// TIA Portal V20 export
FUNCTION_BLOCK "FB_AxisPosition"   // FB411, SCL
{ S7_Optimized_Access := 'TRUE' }
// stored: AutoNumber false, MemoryReserve 100, SetENOAutomatically false
   VAR
      sError { ExternalAccessible := 'False'; ExternalVisible := 'False'; ExternalWritable := 'False'} : Bool;
      sNDR { ExternalAccessible := 'False'; ExternalVisible := 'False'; ExternalWritable := 'False'} : Bool;
      sState { ExternalAccessible := 'False'; ExternalVisible := 'False'; ExternalWritable := 'False'} : Word;
      sAxis01_X : Struct
         "$AA_IM" : LReal;
         "$MA_POS_LIMIT_MINUS" : LReal;
         "$MA_POS_LIMIT_MINUS2" : LReal;
         "$MA_POS_LIMIT_PLUS" : LReal;
         "$MA_POS_LIMIT_PLUS2" : LReal;
         "$MA_JOG_VELO" : LReal;
         "$MA_JOG_VELO_RAPID" : LReal;
         "$MA_MAX_AX_VELO" : LReal;
         "$A1_M_FP_POS4_30600" : LReal;
      END_STRUCT;
      sAxis02_Y : Struct
         "$AA_IM" : LReal;
         "$MA_POS_LIMIT_MINUS" : LReal;
         "$MA_POS_LIMIT_MINUS2" : LReal;
         "$MA_POS_LIMIT_PLUS" : LReal;
         "$MA_POS_LIMIT_PLUS2" : LReal;
         "$MA_JOG_VELO" : LReal;
         "$MA_JOG_VELO_RAPID" : LReal;
         "$MA_MAX_AX_VELO" : LReal;
      END_STRUCT;
      sAxis03_ZM : Struct
         "$AA_IM" : LReal;
         "$MA_POS_LIMIT_MINUS" : LReal;
         "$MA_POS_LIMIT_MINUS2" : LReal;
         "$MA_POS_LIMIT_PLUS" : LReal;
         "$MA_POS_LIMIT_PLUS2" : LReal;
         "$MA_JOG_VELO" : LReal;
         "$MA_JOG_VELO_RAPID" : LReal;
         "$MA_MAX_AX_VELO" : LReal;
      END_STRUCT;
      sAxis04_B : Struct
         "$AA_IM" : LReal;
         "$MA_POS_LIMIT_MINUS" : LReal;
         "$MA_POS_LIMIT_MINUS2" : LReal;
         "$MA_POS_LIMIT_PLUS" : LReal;
         "$MA_POS_LIMIT_PLUS2" : LReal;
         "$MA_JOG_VELO" : LReal;
         "$MA_JOG_VELO_RAPID" : LReal;
         "$MA_MAX_AX_VELO" : LReal;
      END_STRUCT;
      sAxis05_U1 : Struct
         "$AA_IM" : LReal;
         "$MA_POS_LIMIT_MINUS" : LReal;
         "$MA_POS_LIMIT_MINUS2" : LReal;
         "$MA_POS_LIMIT_PLUS" : LReal;
         "$MA_POS_LIMIT_PLUS2" : LReal;
         "$MA_JOG_VELO" : LReal;
         "$MA_JOG_VELO_RAPID" : LReal;
         "$MA_MAX_AX_VELO" : LReal;
      END_STRUCT;
      sAxis06_U2 : Struct
         "$AA_IM" : LReal;
         "$MA_POS_LIMIT_MINUS" : LReal;
         "$MA_POS_LIMIT_MINUS2" : LReal;
         "$MA_POS_LIMIT_PLUS" : LReal;
         "$MA_POS_LIMIT_PLUS2" : LReal;
         "$MA_JOG_VELO" : LReal;
         "$MA_JOG_VELO_RAPID" : LReal;
         "$MA_MAX_AX_VELO" : LReal;
         "$A1_M_FP_POS2_30600" : LReal;
      END_STRUCT;
      sAxis07_V : Struct
         "$AA_IM" : LReal;
         "$MA_POS_LIMIT_MINUS" : LReal;
         "$MA_POS_LIMIT_MINUS2" : LReal;
         "$MA_POS_LIMIT_PLUS" : LReal;
         "$MA_POS_LIMIT_PLUS2" : LReal;
         "$MA_JOG_VELO" : LReal;
         "$MA_JOG_VELO_RAPID" : LReal;
         "$MA_MAX_AX_VELO" : LReal;
      END_STRUCT;
      sAxis08_W : Struct
         "$AA_IM" : LReal;
         "$MA_POS_LIMIT_MINUS" : LReal;
         "$MA_POS_LIMIT_MINUS2" : LReal;
         "$MA_POS_LIMIT_PLUS" : LReal;
         "$MA_POS_LIMIT_PLUS2" : LReal;
         "$MA_JOG_VELO" : LReal;
         "$MA_JOG_VELO_RAPID" : LReal;
         "$MA_MAX_AX_VELO" : LReal;
      END_STRUCT;
      sAxis09_ZL : Struct
         "$AA_IM" : LReal;
         "$MA_POS_LIMIT_MINUS" : LReal;
         "$MA_POS_LIMIT_MINUS2" : LReal;
         "$MA_POS_LIMIT_PLUS" : LReal;
         "$MA_POS_LIMIT_PLUS2" : LReal;
         "$MA_JOG_VELO" : LReal;
         "$MA_JOG_VELO_RAPID" : LReal;
         "$MA_MAX_AX_VELO" : LReal;
      END_STRUCT;
   END_VAR
BEGIN
   REGION Description header 
       //==================================================================================
       // POSALUX Swiss SA / (C) Copyright 2025
       //----------------------------------------------------------------------------------
       // Title: FB_AxisPosition
       // Comment/Function: These function blocks allow reading NC data related to 
       //                   axis positions, references, and speeds from the NC.
       // Author: Fabien WALDT
       // Engineering: TIA Portal v17
       //----------------------------------------------------------------------------------
       // Change log table:
       // Version  | Date     | Expert in charge | Changes applied
       // ---------|----------|------------------|------------------------------------
       // 00.00.01 | 20250423 | WFA              | First released version
       // ==================================================================================
   END_REGION

   REGION Axis 01 X
       "LBP_ReadVar_DB_Axis01_X"(Req := "Clock_10Hz",
                                 NumVar := 8,
                                 Addr1 := "DB_NcVarSelect_AA_IM"."$AA_IM_Axis01_X".token,
                                 Addr2 := "DB_NcVarSelect_MA_POS_LIMIT_MINUS"."$MA_POS_LIMIT_MINUS_Axis01_X".token,
                                 Addr3 := "DB_NcVarSelect_MA_POS_LIMIT_MINUS2"."$MA_POS_LIMIT_MINUS2_Axis01_X".token,
                                 Addr4 := "DB_NcVarSelect_MA_POS_LIMIT_PLUS"."$MA_POS_LIMIT_PLUS_Axis01_X".token,
                                 Addr5 := "DB_NcVarSelect_MA_POS_LIMIT_PLUS2"."$MA_POS_LIMIT_PLUS2_Axis01_X".token,
                                 Addr6 := "DB_NcVarSelect_MA_JOG_VELO"."$MA_JOG_VELO_Axis01_X".token,
                                 Addr7 := "DB_NcVarSelect_MA_JOG_VELO_RAPID"."$MA_JOG_VELO_RAPID_Axis01_X".token,
                                 Addr8 := "DB_NcVarSelect_M_MAX_AX_VELO"."$MA_JOG_VELO_Axis01_X".token,
                                 Error => #sError,
                                 NDR => #sNDR,
                                 State => #sState,
                                 RD1 := #sAxis01_X."$AA_IM",
                                 RD2 := #sAxis01_X."$MA_POS_LIMIT_MINUS",
                                 RD3 := #sAxis01_X."$MA_POS_LIMIT_MINUS2",
                                 RD4 := #sAxis01_X."$MA_POS_LIMIT_PLUS",
                                 RD5 := #sAxis01_X."$MA_POS_LIMIT_PLUS2",
                                 RD6 := #sAxis01_X."$MA_JOG_VELO",
                                 RD7 := #sAxis01_X."$MA_JOG_VELO_RAPID",
                                 RD8 := #sAxis01_X."$MA_MAX_AX_VELO");
   END_REGION

   REGION Axis 02 Y
       "LBP_ReadVar_DB_Axis02_Y"(Req := "Clock_10Hz",
                                 NumVar := 8,
                                 Addr1 := "DB_NcVarSelect_AA_IM"."$AA_IM_Axis02_Y".token,
                                 Addr2 := "DB_NcVarSelect_MA_POS_LIMIT_MINUS"."$MA_POS_LIMIT_MINUS_Axis02_Y".token,
                                 Addr3 := "DB_NcVarSelect_MA_POS_LIMIT_MINUS2"."$MA_POS_LIMIT_MINUS2_Axis02_Y".token,
                                 Addr4 := "DB_NcVarSelect_MA_POS_LIMIT_PLUS"."$MA_POS_LIMIT_PLUS_Axis02_Y".token,
                                 Addr5 := "DB_NcVarSelect_MA_POS_LIMIT_PLUS2"."$MA_POS_LIMIT_PLUS2_Axis02_Y".token,
                                 Addr6 := "DB_NcVarSelect_MA_JOG_VELO"."$MA_JOG_VELO_Axis02_Y".token,
                                 Addr7 := "DB_NcVarSelect_MA_JOG_VELO_RAPID"."$MA_JOG_VELO_RAPID_Axis02_Y".token,
                                 Addr8 := "DB_NcVarSelect_M_MAX_AX_VELO"."$MA_JOG_VELO_Axis02_Y".token,
                                 Error => #sError,
                                 NDR => #sNDR,
                                 State => #sState,
                                 RD1 := #sAxis02_Y."$AA_IM",
                                 RD2 := #sAxis02_Y."$MA_POS_LIMIT_MINUS",
                                 RD3 := #sAxis02_Y."$MA_POS_LIMIT_MINUS2",
                                 RD4 := #sAxis02_Y."$MA_POS_LIMIT_PLUS",
                                 RD5 := #sAxis02_Y."$MA_POS_LIMIT_PLUS2",
                                 RD6 := #sAxis02_Y."$MA_JOG_VELO",
                                 RD7 := #sAxis02_Y."$MA_JOG_VELO_RAPID",
                                 RD8 := #sAxis02_Y."$MA_MAX_AX_VELO");
   END_REGION

   REGION Axis 03 ZM
       "LBP_ReadVar_DB_Axis03_ZM"(Req := "Clock_10Hz",
                                  NumVar := 8,
                                  Addr1 := "DB_NcVarSelect_AA_IM"."$AA_IM_Axis03_ZM".token,
                                  Addr2 := "DB_NcVarSelect_MA_POS_LIMIT_MINUS"."$MA_POS_LIMIT_MINUS_Axis03_ZM".token,
                                  Addr3 := "DB_NcVarSelect_MA_POS_LIMIT_MINUS2"."$MA_POS_LIMIT_MINUS2_Axis03_ZM".token,
                                  Addr4 := "DB_NcVarSelect_MA_POS_LIMIT_PLUS"."$MA_POS_LIMIT_PLUS_Axis03_ZM".token,
                                  Addr5 := "DB_NcVarSelect_MA_POS_LIMIT_PLUS2"."$MA_POS_LIMIT_PLUS2_Axis03_ZM".token,
                                  Addr6 := "DB_NcVarSelect_MA_JOG_VELO"."$MA_JOG_VELO_Axis03_ZM".token,
                                  Addr7 := "DB_NcVarSelect_MA_JOG_VELO_RAPID"."$MA_JOG_VELO_RAPID_Axis03_ZM".token,
                                  Addr8 := "DB_NcVarSelect_M_MAX_AX_VELO"."$MA_JOG_VELO_Axis03_ZM".token,
                                  Error => #sError,
                                  NDR => #sNDR,
                                  State => #sState,
                                  RD1 := #sAxis03_ZM."$AA_IM",
                                  RD2 := #sAxis03_ZM."$MA_POS_LIMIT_MINUS",
                                  RD3 := #sAxis03_ZM."$MA_POS_LIMIT_MINUS2",
                                  RD4 := #sAxis03_ZM."$MA_POS_LIMIT_PLUS",
                                  RD5 := #sAxis03_ZM."$MA_POS_LIMIT_PLUS2",
                                  RD6 := #sAxis03_ZM."$MA_JOG_VELO",
                                  RD7 := #sAxis03_ZM."$MA_JOG_VELO_RAPID",
                                  RD8 := #sAxis03_ZM."$MA_MAX_AX_VELO");
   END_REGION

   REGION Axis 04 B
       "LBP_ReadVar_DB_Axis04_B"(Req := "Clock_10Hz",
                                 NumVar := 8,
                                 Addr1 := "DB_NcVarSelect_AA_IM"."$AA_IM_Axis04_B".token,
                                 Addr2 := "DB_NcVarSelect_MA_POS_LIMIT_MINUS"."$MA_POS_LIMIT_MINUS_Axis04_B".token,
                                 Addr3 := "DB_NcVarSelect_MA_POS_LIMIT_MINUS2"."$MA_POS_LIMIT_MINUS2_Axis04_B".token,
                                 Addr4 := "DB_NcVarSelect_MA_POS_LIMIT_PLUS"."$MA_POS_LIMIT_PLUS_Axis04_B".token,
                                 Addr5 := "DB_NcVarSelect_MA_POS_LIMIT_PLUS2"."$MA_POS_LIMIT_PLUS2_Axis04_B".token,
                                 Addr6 := "DB_NcVarSelect_MA_JOG_VELO"."$MA_JOG_VELO_Axis04_B".token,
                                 Addr7 := "DB_NcVarSelect_MA_JOG_VELO_RAPID"."$MA_JOG_VELO_RAPID_Axis04_B".token,
                                 Addr8 := "DB_NcVarSelect_M_MAX_AX_VELO"."$MA_JOG_VELO_Axis04_B".token,
                                 Error => #sError,
                                 NDR => #sNDR,
                                 State => #sState,
                                 RD1 := #sAxis04_B."$AA_IM",
                                 RD2 := #sAxis04_B."$MA_POS_LIMIT_MINUS",
                                 RD3 := #sAxis04_B."$MA_POS_LIMIT_MINUS2",
                                 RD4 := #sAxis04_B."$MA_POS_LIMIT_PLUS",
                                 RD5 := #sAxis04_B."$MA_POS_LIMIT_PLUS2",
                                 RD6 := #sAxis04_B."$MA_JOG_VELO",
                                 RD7 := #sAxis04_B."$MA_JOG_VELO_RAPID",
                                 RD8 := #sAxis04_B."$MA_MAX_AX_VELO");
   END_REGION

   REGION Axis 05 U1
       "LBP_ReadVar_DB_Axis05_U1"(Req := NOT "Clock_10Hz",
                                  NumVar := 8,
                                  Addr1 := "DB_NcVarSelect_AA_IM"."$AA_IM_Axis05_U1".token,
                                  Addr2 := "DB_NcVarSelect_MA_POS_LIMIT_MINUS"."$MA_POS_LIMIT_MINUS_Axis05_U1".token,
                                  Addr3 := "DB_NcVarSelect_MA_POS_LIMIT_MINUS2"."$MA_POS_LIMIT_MINUS2_Axis05_U1".token,
                                  Addr4 := "DB_NcVarSelect_MA_POS_LIMIT_PLUS"."$MA_POS_LIMIT_PLUS_Axis05_U1".token,
                                  Addr5 := "DB_NcVarSelect_MA_POS_LIMIT_PLUS2"."$MA_POS_LIMIT_PLUS2_Axis05_U1".token,
                                  Addr6 := "DB_NcVarSelect_MA_JOG_VELO"."$MA_JOG_VELO_Axis05_U1".token,
                                  Addr7 := "DB_NcVarSelect_MA_JOG_VELO_RAPID"."$MA_JOG_VELO_RAPID_Axis05_U1".token,
                                  Addr8 := "DB_NcVarSelect_M_MAX_AX_VELO"."$MA_JOG_VELO_Axis05_U1".token,
                                  Error => #sError,
                                  NDR => #sNDR,
                                  State => #sState,
                                  RD1 := #sAxis05_U1."$AA_IM",
                                  RD2 := #sAxis05_U1."$MA_POS_LIMIT_MINUS",
                                  RD3 := #sAxis05_U1."$MA_POS_LIMIT_MINUS2",
                                  RD4 := #sAxis05_U1."$MA_POS_LIMIT_PLUS",
                                  RD5 := #sAxis05_U1."$MA_POS_LIMIT_PLUS2",
                                  RD6 := #sAxis05_U1."$MA_JOG_VELO",
                                  RD7 := #sAxis05_U1."$MA_JOG_VELO_RAPID",
                                  RD8 := #sAxis05_U1."$MA_MAX_AX_VELO");
   END_REGION

   REGION Axis 06 U2
       "LBP_ReadVar_DB_Axis06_U2"(Req := NOT "Clock_10Hz",
                                  NumVar := 8,
                                  Addr1 := "DB_NcVarSelect_AA_IM"."$AA_IM_Axis06_U2".token,
                                  Addr2 := "DB_NcVarSelect_MA_POS_LIMIT_MINUS"."$MA_POS_LIMIT_MINUS_Axis06_U2".token,
                                  Addr3 := "DB_NcVarSelect_MA_POS_LIMIT_MINUS2"."$MA_POS_LIMIT_MINUS2_Axis06_U2".token,
                                  Addr4 := "DB_NcVarSelect_MA_POS_LIMIT_PLUS"."$MA_POS_LIMIT_PLUS_Axis06_U2".token,
                                  Addr5 := "DB_NcVarSelect_MA_POS_LIMIT_PLUS2"."$MA_POS_LIMIT_PLUS2_Axis06_U2".token,
                                  Addr6 := "DB_NcVarSelect_MA_JOG_VELO"."$MA_JOG_VELO_Axis06_U2".token,
                                  Addr7 := "DB_NcVarSelect_MA_JOG_VELO_RAPID"."$MA_JOG_VELO_RAPID_Axis06_U2".token,
                                  Addr8 := "DB_NcVarSelect_M_MAX_AX_VELO"."$MA_JOG_VELO_Axis06_U2".token,
                                  Error => #sError,
                                  NDR => #sNDR,
                                  State => #sState,
                                  RD1 := #sAxis06_U2."$AA_IM",
                                  RD2 := #sAxis06_U2."$MA_POS_LIMIT_MINUS",
                                  RD3 := #sAxis06_U2."$MA_POS_LIMIT_MINUS2",
                                  RD4 := #sAxis06_U2."$MA_POS_LIMIT_PLUS",
                                  RD5 := #sAxis06_U2."$MA_POS_LIMIT_PLUS2",
                                  RD6 := #sAxis06_U2."$MA_JOG_VELO",
                                  RD7 := #sAxis06_U2."$MA_JOG_VELO_RAPID",
                                  RD8 := #sAxis06_U2."$MA_MAX_AX_VELO");
   END_REGION

   REGION Axis 07 V
       "LBP_ReadVar_DB_Axis07_V"(Req := NOT "Clock_10Hz",
                                 NumVar := 8,
                                 Addr1 := "DB_NcVarSelect_AA_IM"."$AA_IM_Axis07_V".token,
                                 Addr2 := "DB_NcVarSelect_MA_POS_LIMIT_MINUS"."$MA_POS_LIMIT_MINUS_Axis07_V".token,
                                 Addr3 := "DB_NcVarSelect_MA_POS_LIMIT_MINUS2"."$MA_POS_LIMIT_MINUS2_Axis07_V".token,
                                 Addr4 := "DB_NcVarSelect_MA_POS_LIMIT_PLUS"."$MA_POS_LIMIT_PLUS_Axis07_V".token,
                                 Addr5 := "DB_NcVarSelect_MA_POS_LIMIT_PLUS2"."$MA_POS_LIMIT_PLUS2_Axis07_V".token,
                                 Addr6 := "DB_NcVarSelect_MA_JOG_VELO"."$MA_JOG_VELO_Axis07_V".token,
                                 Addr7 := "DB_NcVarSelect_MA_JOG_VELO_RAPID"."$MA_JOG_VELO_RAPID_Axis07_V".token,
                                 Addr8 := "DB_NcVarSelect_M_MAX_AX_VELO"."$MA_JOG_VELO_Axis07_V".token,
                                 Error => #sError,
                                 NDR => #sNDR,
                                 State => #sState,
                                 RD1 := #sAxis07_V."$AA_IM",
                                 RD2 := #sAxis07_V."$MA_POS_LIMIT_MINUS",
                                 RD3 := #sAxis07_V."$MA_POS_LIMIT_MINUS2",
                                 RD4 := #sAxis07_V."$MA_POS_LIMIT_PLUS",
                                 RD5 := #sAxis07_V."$MA_POS_LIMIT_PLUS2",
                                 RD6 := #sAxis07_V."$MA_JOG_VELO",
                                 RD7 := #sAxis07_V."$MA_JOG_VELO_RAPID",
                                 RD8 := #sAxis07_V."$MA_MAX_AX_VELO");
   END_REGION

   REGION Axis 08 W
       "LBP_ReadVar_DB_Axis08_W"(Req := NOT "Clock_10Hz",
                                 NumVar := 8,
                                 Addr1 := "DB_NcVarSelect_AA_IM"."$AA_IM_Axis08_W".token,
                                 Addr2 := "DB_NcVarSelect_MA_POS_LIMIT_MINUS"."$MA_POS_LIMIT_MINUS_Axis08_W".token,
                                 Addr3 := "DB_NcVarSelect_MA_POS_LIMIT_MINUS2"."$MA_POS_LIMIT_MINUS2_Axis08_W".token,
                                 Addr4 := "DB_NcVarSelect_MA_POS_LIMIT_PLUS"."$MA_POS_LIMIT_PLUS_Axis08_W".token,
                                 Addr5 := "DB_NcVarSelect_MA_POS_LIMIT_PLUS2"."$MA_POS_LIMIT_PLUS2_Axis08_W".token,
                                 Addr6 := "DB_NcVarSelect_MA_JOG_VELO"."$MA_JOG_VELO_Axis08_W".token,
                                 Addr7 := "DB_NcVarSelect_MA_JOG_VELO_RAPID"."$MA_JOG_VELO_RAPID_Axis08_W".token,
                                 Addr8 := "DB_NcVarSelect_M_MAX_AX_VELO"."$MA_JOG_VELO_Axis08_W".token,
                                 Error => #sError,
                                 NDR => #sNDR,
                                 State => #sState,
                                 RD1 := #sAxis08_W."$AA_IM",
                                 RD2 := #sAxis08_W."$MA_POS_LIMIT_MINUS",
                                 RD3 := #sAxis08_W."$MA_POS_LIMIT_MINUS2",
                                 RD4 := #sAxis08_W."$MA_POS_LIMIT_PLUS",
                                 RD5 := #sAxis08_W."$MA_POS_LIMIT_PLUS2",
                                 RD6 := #sAxis08_W."$MA_JOG_VELO",
                                 RD7 := #sAxis08_W."$MA_JOG_VELO_RAPID",
                                 RD8 := #sAxis08_W."$MA_MAX_AX_VELO");
   END_REGION

   REGION Axis 09 ZL
       "LBP_ReadVar_DB_Axis09_ZL"(Req := "Clock_10Hz",
                                  NumVar := 8,
                                  Addr1 := "DB_NcVarSelect_AA_IM"."$AA_IM_Axis09_ZL".token,
                                  Addr2 := "DB_NcVarSelect_MA_POS_LIMIT_MINUS"."$MA_POS_LIMIT_MINUS_Axis09_ZL".token,
                                  Addr3 := "DB_NcVarSelect_MA_POS_LIMIT_MINUS2"."$MA_POS_LIMIT_MINUS2_Axis09_ZL".token,
                                  Addr4 := "DB_NcVarSelect_MA_POS_LIMIT_PLUS"."$MA_POS_LIMIT_PLUS_Axis09_ZL".token,
                                  Addr5 := "DB_NcVarSelect_MA_POS_LIMIT_PLUS2"."$MA_POS_LIMIT_PLUS2_Axis09_ZL".token,
                                  Addr6 := "DB_NcVarSelect_MA_JOG_VELO"."$MA_JOG_VELO_Axis09_ZL".token,
                                  Addr7 := "DB_NcVarSelect_MA_JOG_VELO_RAPID"."$MA_JOG_VELO_RAPID_Axis09_ZL".token,
                                  Addr8 := "DB_NcVarSelect_M_MAX_AX_VELO"."$MA_JOG_VELO_Axis09_ZL".token,
                                  Error => #sError,
                                  NDR => #sNDR,
                                  State => #sState,
                                  RD1 := #sAxis09_ZL."$AA_IM",
                                  RD2 := #sAxis09_ZL."$MA_POS_LIMIT_MINUS",
                                  RD3 := #sAxis09_ZL."$MA_POS_LIMIT_MINUS2",
                                  RD4 := #sAxis09_ZL."$MA_POS_LIMIT_PLUS",
                                  RD5 := #sAxis09_ZL."$MA_POS_LIMIT_PLUS2",
                                  RD6 := #sAxis09_ZL."$MA_JOG_VELO",
                                  RD7 := #sAxis09_ZL."$MA_JOG_VELO_RAPID",
                                  RD8 := #sAxis09_ZL."$MA_MAX_AX_VELO");
    END_REGION
END_FUNCTION_BLOCK
